PROGRAM MAIN
VAR
END_VAR

GVL.rY := GVL.rY + 0.1;
GVL.rX := GVL.rY;

IF GVL.rY > 100.0 THEN
	GVL.rY := 0;
END_IF

END_PROGRAM

(* stored: Version 1.1.0.1, ProductVersion 3.1.4024.13
   POU MAIN: Id {5e7b9ce6-4fbf-403c-b63a-498716304f58}, SpecialFunc None *)
